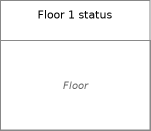
VISUALIZATION Screen1  // 151x131
    Frame (0,40 151x91)
        shows Floor(LS_Floor := MAIN.LS_Floor[1])
        OnMouseClick: change screen: Previous 
    Label (0,0 150x30), "Floor 1 status"
END_VISUALIZATION

(* stored: Version 1.1.0.1, ProductVersion 3.1.4024.11
   Visu Screen1: Id {f5a3fa43-64ec-4dd5-9396-fe78d897518c} *)
